// TIA Portal V20 export
DATA_BLOCK "Fault_DB"   // DB304
// stored: AutoNumber false, InstanceOfName Fault, InstanceOfType FB
"Fault"
   // VAR
   //    Var : "TypeVar";
   //    T : Array[1..16] of IEC_TIMER;
   //    ErrSafetyModule { ExternalAccessible := 'False'; ExternalVisible := 'False'; ExternalWritable := 'False'} : Bool;
   // END_VAR
BEGIN
END_DATA_BLOCK
